Yaskawa INFORM job: TRIANGULO20250509100134.JBI

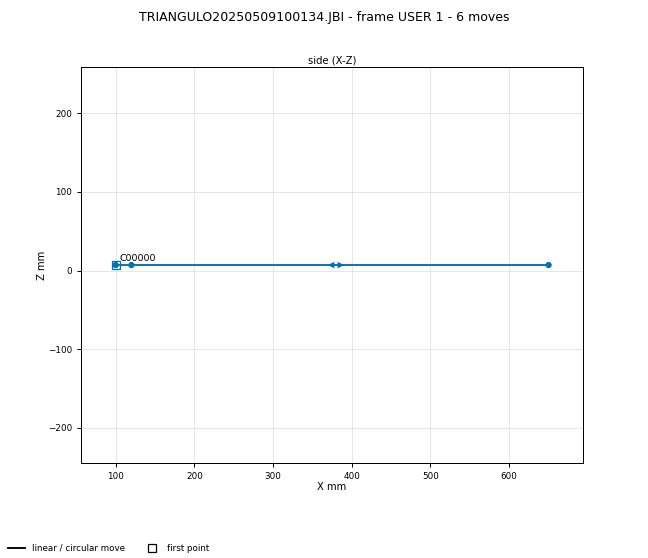
[picture p0: tool path of TRIANGULO20250509100134.JBI in frame USER 1, 6 of 6 moves have a stored position in this frame; points joined in program order, loops and branches not executed]
/JOB
//NAME TRIANGUL
//POS
///NPOS 6,0,0,0,0,0
///USER 1
///TOOL 0
///POSTYPE USER
///RECTAN
///RCONF 1,0,0,0,0,0,0,0,0,0,0,0,0,0,0,0,0,0,0,0,0,0,0,0
C00000=100,100,7,0,0,0
C00001=120,100,7,0,0,0
C00002=120,100,7,0,0,0
C00003=650,100,7,0,0,0
C00004=650,100,7,0,0,0
C00005=100,100,7,0,0,0
//INST
///DATE 2025/05/09 10:01
///ATTR SC,RW,RJ
////FRAME USER 1
///GROUP1 RB1
NOP
MOVJ C00000 VJ=0.78
MOVL C00001 V=30.0
MOVL C00002 V=30.0
MOVL C00003 V=30.0
MOVL C00004 V=30.0
MOVL C00005 V=30.0
END
